// TIA Portal V17 export
// export: Created 2022-09-15T00:24:46.0287989Z, ExportSetting WithDefaults, DisplayName Totally Integrated Automation Portal, DisplayVersion V17, DisplayName TIA Portal Openness, DisplayVersion V17, DisplayName TIA Portal Version Control Interface, DisplayVersion V17, DisplayName SINAMICS Startdrive Advanced, DisplayVersion V17 Update1, DisplayName SINAMICS Startdrive G110M, G120, G120C, G120D, G120P, G115D, DisplayVersion V17 Update1, DisplayName SINAMICS Startdrive G130, G150, S120, S150, SINAMICS MV, S210, DisplayVersion V17 Update1, DisplayName STEP 7 Professional, DisplayVersion V17, DisplayName STEP 7 Safety, DisplayVersion V17, DisplayName WinCC Advanced / Unified PC, DisplayVersion V17
VAR_GLOBAL   // PLC tag table "Default tag table"
   AX_4_Actor_Interface_AddressIn AT %I356.0 : "PD_TEL105_IN";
   AX_4_Actor_Interface_AddressOut AT %Q356.0 : "PD_TEL105_OUT";
   AX_4_Actor_Interface_TorqueDataAddressIn AT %I382.0 : "PD_TEL750_IN";
   AX_4_Actor_Interface_TorqueDataAddressOut AT %Q382.0 : "PD_TEL750_OUT";
   AX_3_Actor_Interface_AddressIn AT %I324.0 : "PD_TEL105_IN";
   AX_3_Actor_Interface_AddressOut AT %Q324.0 : "PD_TEL105_OUT";
   AX_3_Actor_Interface_TorqueDataAddressIn AT %I350.0 : "PD_TEL750_IN";
   AX_3_Actor_Interface_TorqueDataAddressOut AT %Q350.0 : "PD_TEL750_OUT";
   AX_2_Actor_Interface_AddressIn AT %I292.0 : "PD_TEL105_IN";
   AX_2_Actor_Interface_AddressOut AT %Q292.0 : "PD_TEL105_OUT";
   AX_2_Actor_Interface_TorqueDataAddressIn AT %I318.0 : "PD_TEL750_IN";
   AX_2_Actor_Interface_TorqueDataAddressOut AT %Q318.0 : "PD_TEL750_OUT";
   AX_1_Actor_Interface_AddressIn AT %I260.0 : "PD_TEL105_IN";
   AX_1_Actor_Interface_AddressOut AT %Q260.0 : "PD_TEL105_OUT";
   AX_1_Actor_Interface_TorqueDataAddressIn AT %I286.0 : "PD_TEL750_IN";
   AX_1_Actor_Interface_TorqueDataAddressOut AT %Q286.0 : "PD_TEL750_OUT";
   SpeedAxis_Actor_Interface_AddressIn AT %I288.0 : "PD_TEL1_IN";
   SpeedAxis_Actor_Interface_AddressOut AT %Q390.0 : "PD_TEL1_OUT";
   Tag_1 AT %M0.0 : Bool;
   Tag_2 AT %M0.1 : Bool;
   Tag_3 AT %M0.2 : Bool;
   Tag_4 AT %M0.3 : Bool;
END_VAR
